{attribute 'linkalways'}
{attribute 'hide_all_locals'}
FUNCTION_BLOCK ValueLword EXTENDS ValueLwordRead IMPLEMENTS Value
VAR
END_VAR

METHOD SetFromType : BOOL
VAR_INPUT
	source : __SYSTEM.AnyType;
END_VAR
SetFromType := ConvertAnyType(source, thisAnyType);
END_METHOD

METHOD SetFromString : BOOL
VAR_INPUT
	value : T_MaxString;
END_VAR
thisValue := STRING_TO_LWORD(value);

SetFromString := TRUE;
END_METHOD

METHOD Set : BOOL
VAR_INPUT
	source : ANY;
END_VAR
Set := ConvertAnyType(source, thisAnyType);
END_METHOD

END_FUNCTION_BLOCK

(* stored: Version 1.1.0.1
   POU ValueLword: Id {a01edb43-74e5-46d5-9620-42e78ed6bfd6}, SpecialFunc None
   Method SetFromType: Id {51675e0e-f5c6-417f-838f-24afe5002e38}
   Method SetFromString: Id {2b6e1fb1-ea84-451f-be8a-755063524fbd}
   Method Set: Id {99ffa13b-2144-44a9-8171-ff18826c5e1f} *)
